// TIA Portal V19 export
DATA_BLOCK "RollformerLubr"   // DB140
// stored: InstanceOfName RollformerLubr_FB, InstanceOfType FB
"RollformerLubr_FB"
   // VAR_INPUT
   //    AreaInterface : "AreaInterface";
   // END_VAR
   // VAR_OUTPUT
   //    MachineInterface : "MachineInterface";
   // END_VAR
   // VAR
   //    Pump : "Lubr_Motor";
   //    Valves1 : "Lubr_Valve";
   //    Valves2 { S7_SetPoint := 'True'} : "Lubr_Valve";
   //    Valves3 { S7_SetPoint := 'True'} : "Lubr_Valve";
   // END_VAR
BEGIN
   AreaInterface.EStop := FALSE;
   AreaInterface.Man := TRUE;
   AreaInterface.Aut := FALSE;
   AreaInterface.Cycle := FALSE;
   AreaInterface.StopInPhase := FALSE;
   AreaInterface.StopProgrammed := FALSE;
   AreaInterface.RstAlarms := FALSE;
   AreaInterface.ManOneShot := FALSE;
   AreaInterface.AutOneShot := FALSE;
   AreaInterface.CycleOneShot := FALSE;
   AreaInterface.CheckAutReady := FALSE;
   MachineInterface.AutReady := FALSE;
   MachineInterface.Aborting := FALSE;
   MachineInterface.AckStopInPhase := FALSE;
   MachineInterface.AckStopProgrammed := FALSE;
   MachineInterface.MotionsStandStill := TRUE;
   MachineInterface.AlarmsPresence := FALSE;
   MachineInterface.WarningPresence := FALSE;
   Pump.DataIn.PbManualLubr := FALSE;
   Pump.DataIn.LubrRotationFbk := FALSE;
   Pump.DataIn.SensorLevel := TRUE;
   Pump.DataIn.MotorFdbkRunning := FALSE;
   Pump.DataIn.MotorThermalProtection := FALSE;
   Pump.ValveCycleTimeOut := T#5M;
   Pump.Simulation := FALSE;
   Pump.RunContactor := FALSE;
   Pump.Ctrl.RunReq := FALSE;
   Pump.Sts.OldValve := 1;
   Pump.Alarm.RotationFeedback := FALSE;
   Pump.Alarm.LowLevelLubrication := FALSE;
   Pump.Alarm.MotorAlr.ThermalProtection := FALSE;
   Pump.Alarm.MotorAlr.Feedback := FALSE;
   Pump.HMI.Alarm := FALSE;
   Pump.HMI.Running := FALSE;
   Pump.LubrInterface.Sts.PumpType := 0;
   Pump.LubrInterface.Sts.Running := FALSE;
   Pump.LubrInterface.Sts.Error := FALSE;
   Pump.LubrInterface.Ctrl.RstAlarms := FALSE;
   Pump.LubrInterface.Ctrl.WorkReq := FALSE;
   Pump.LubrInterface.ValveChain.ActualValve := 4;
   Pump.LubrInterface.ValveChain.MaxValve := 3;
   Pump.tonRotationON.PT := T#0MS;
   Pump.tonRotationON.IN := FALSE;
   Pump.tonRotationOFF.PT := T#0MS;
   Pump.tonRotationOFF.IN := FALSE;
   Pump.tonLowLevel.PT := T#0MS;
   Pump.tonLowLevel.IN := FALSE;
   Pump.ValveChianTimeOut.PT := T#5M;
   Pump.ValveChianTimeOut.IN := TRUE;
   Pump.LubrMotor.MotorCtrl.SafeStop := FALSE;
   Pump.LubrMotor.MotorCtrl.Rst := FALSE;
   Pump.LubrMotor.MotorCtrl.Run := FALSE;
   Pump.LubrMotor.ThermalProtection := FALSE;
   Pump.LubrMotor.FdbkRunning := FALSE;
   Pump.LubrMotor.FeedbackTimeout := T#500MS;
   Pump.LubrMotor.Simulation := FALSE;
   Pump.LubrMotor.MotorSts.AlarmPresence := FALSE;
   Pump.LubrMotor.MotorSts.RunPermitted := TRUE;
   Pump.LubrMotor.MotorSts.Running := FALSE;
   Pump.LubrMotor.Contactor := FALSE;
   Pump.LubrMotor.DelayContactorFeedbackON.PT := T#500MS;
   Pump.LubrMotor.DelayContactorFeedbackON.IN := FALSE;
   Pump.LubrMotor.Ctrl_RunContactor := FALSE;
   Valves1.AreaInterface.EStop := FALSE;
   Valves1.AreaInterface.Man := TRUE;
   Valves1.AreaInterface.Aut := FALSE;
   Valves1.AreaInterface.Cycle := FALSE;
   Valves1.AreaInterface.StopInPhase := FALSE;
   Valves1.AreaInterface.StopProgrammed := FALSE;
   Valves1.AreaInterface.RstAlarms := FALSE;
   Valves1.AreaInterface.ManOneShot := FALSE;
   Valves1.AreaInterface.AutOneShot := FALSE;
   Valves1.AreaInterface.CycleOneShot := FALSE;
   Valves1.AreaInterface.CheckAutReady := FALSE;
   Valves1.DataIn.PbStartLubr := FALSE;
   Valves1.DataIn.PbStopLubr := FALSE;
   Valves1.DataIn.CycleFbk := FALSE;
   Valves1.DataIn.ConnectorPlugged := TRUE;
   Valves1.CIn.LubrEnable := FALSE;
   Valves1.CIn.ActualPosition := 324862.052;
   Valves1.CIn.OperationDone := FALSE;
   Valves1.Config.WorkMode := 2;
   Valves1.Config.CounterMode := 0;
   Valves1.Config.ValveType := 1;
   Valves1.Config.ManualCmdTimeOut := T#5M;
   Valves1.Simulation := FALSE;
   Valves1.MachineInterface.AutReady := FALSE;
   Valves1.MachineInterface.Aborting := FALSE;
   Valves1.MachineInterface.AckStopInPhase := FALSE;
   Valves1.MachineInterface.AckStopProgrammed := FALSE;
   Valves1.MachineInterface.MotionsStandStill := TRUE;
   Valves1.MachineInterface.AlarmsPresence := FALSE;
   Valves1.MachineInterface.WarningPresence := FALSE;
   Valves1.COut.LubrReq := FALSE;
   Valves1.ValveCmd := FALSE;
   Valves1.Ctrl.ManualReq := FALSE;
   Valves1.Ctrl.AutomaticReq := FALSE;
   Valves1.Ctrl.LubrReq := FALSE;
   Valves1.Ctrl.ValveCmd := FALSE;
   Valves1.Sts.EstopDelayed := FALSE;
   Valves1.Sts.ValveEnabled := TRUE;
   Valves1.Sts.WorkEnable := TRUE;
   Valves1.Sts.CycleDone := FALSE;
   Valves1.Sts.LastFeed := 324862.052;
   Valves1.Sts.IsStandstill := TRUE;
   Valves1.Sts.AlarmsPresence := FALSE;
   Valves1.Sts.WarningsPresence := FALSE;
   Valves1.Alarm.CycleFeedback := FALSE;
   Valves1.Alarm.ConnectorNotPlugged := FALSE;
   Valves1.Alarm.ConfigError := FALSE;
   Valves1.Warning.SystemNotON := FALSE;
   Valves1.HMI.ManReq := FALSE;
   Valves1.HMI.AutoReq := FALSE;
   Valves1.HMI.Running := FALSE;
   Valves1.HMI.Alarm := FALSE;
   Valves1.HMI.ActualWorkTime := T#0MS;
   Valves1.tonEStopDelayed.PT := T#0MS;
   Valves1.tonEStopDelayed.IN := FALSE;
   Valves1.tonCycleDoneON.PT := T#0MS;
   Valves1.tonCycleDoneON.IN := FALSE;
   Valves1.tonCycleDoneOFF.PT := T#0MS;
   Valves1.tonCycleDoneOFF.IN := FALSE;
   Valves1.tonManualCycleReset.PT := T#5M;
   Valves1.tonManualCycleReset.IN := FALSE;
   Valves1.tonValveOn.PT := T#1S;
   Valves1.tonValveOn.IN := FALSE;
   Valves1.tonValveOff.PT := T#1S;
   Valves1.tonValveOff.IN := TRUE;
   Valves1.tonWorkTime.IN := FALSE;
   Valves1.tonWorkTime.ENA := FALSE;
   Valves1.tonWorkTime.PT := T#0MS;
   Valves1.tonWorkTime.Q := TRUE;
   Valves1.tonWorkTime.ET := T#0MS;
   Valves1.tonWorkTime.ton.PT := T#0MS;
   Valves1.tonWorkTime.ton.IN := FALSE;
   Valves1.tonWorkTime.LocalPT := T#0MS;
   Valves1.tonWorkTime.AuxSavePT := FALSE;
   Valves1.Aux_PbStartLubr := FALSE;
   Valves1.Pe_PbStartLubr := FALSE;
   Valves1.Aux_CyckeFkb := FALSE;
   Valves1.Pe_CycleFbk := FALSE;
   Valves1.Aux_OpDone := FALSE;
   Valves1.Pe_OpDone := FALSE;
   Valves1.Aux_ValveCount := TRUE;
   Valves1.Pe_ValveCount := FALSE;
   Valves2.AreaInterface.EStop := FALSE;
   Valves2.AreaInterface.Man := TRUE;
   Valves2.AreaInterface.Aut := FALSE;
   Valves2.AreaInterface.Cycle := FALSE;
   Valves2.AreaInterface.StopInPhase := FALSE;
   Valves2.AreaInterface.StopProgrammed := FALSE;
   Valves2.AreaInterface.RstAlarms := FALSE;
   Valves2.AreaInterface.ManOneShot := FALSE;
   Valves2.AreaInterface.AutOneShot := FALSE;
   Valves2.AreaInterface.CycleOneShot := FALSE;
   Valves2.AreaInterface.CheckAutReady := FALSE;
   Valves2.DataIn.PbStartLubr := FALSE;
   Valves2.DataIn.PbStopLubr := FALSE;
   Valves2.DataIn.CycleFbk := FALSE;
   Valves2.DataIn.ConnectorPlugged := TRUE;
   Valves2.CIn.LubrEnable := FALSE;
   Valves2.CIn.ActualPosition := 324862.052;
   Valves2.CIn.OperationDone := FALSE;
   Valves2.Config.WorkMode := 2;
   Valves2.Config.CounterMode := 0;
   Valves2.Config.ValveType := 1;
   Valves2.Config.ManualCmdTimeOut := T#5M;
   Valves2.Simulation := FALSE;
   Valves2.MachineInterface.AutReady := FALSE;
   Valves2.MachineInterface.Aborting := FALSE;
   Valves2.MachineInterface.AckStopInPhase := FALSE;
   Valves2.MachineInterface.AckStopProgrammed := FALSE;
   Valves2.MachineInterface.MotionsStandStill := TRUE;
   Valves2.MachineInterface.AlarmsPresence := FALSE;
   Valves2.MachineInterface.WarningPresence := FALSE;
   Valves2.COut.LubrReq := FALSE;
   Valves2.ValveCmd := FALSE;
   Valves2.Ctrl.ManualReq := FALSE;
   Valves2.Ctrl.AutomaticReq := FALSE;
   Valves2.Ctrl.LubrReq := FALSE;
   Valves2.Ctrl.ValveCmd := FALSE;
   Valves2.Sts.EstopDelayed := FALSE;
   Valves2.Sts.ValveEnabled := TRUE;
   Valves2.Sts.WorkEnable := TRUE;
   Valves2.Sts.CycleDone := FALSE;
   Valves2.Sts.LastFeed := 324862.052;
   Valves2.Sts.IsStandstill := TRUE;
   Valves2.Sts.AlarmsPresence := FALSE;
   Valves2.Sts.WarningsPresence := FALSE;
   Valves2.Alarm.CycleFeedback := FALSE;
   Valves2.Alarm.ConnectorNotPlugged := FALSE;
   Valves2.Alarm.ConfigError := FALSE;
   Valves2.Warning.SystemNotON := FALSE;
   Valves2.HMI.ManReq := FALSE;
   Valves2.HMI.AutoReq := FALSE;
   Valves2.HMI.Running := FALSE;
   Valves2.HMI.Alarm := FALSE;
   Valves2.HMI.ActualWorkTime := T#0MS;
   Valves2.tonEStopDelayed.PT := T#0MS;
   Valves2.tonEStopDelayed.IN := FALSE;
   Valves2.tonCycleDoneON.PT := T#0MS;
   Valves2.tonCycleDoneON.IN := FALSE;
   Valves2.tonCycleDoneOFF.PT := T#0MS;
   Valves2.tonCycleDoneOFF.IN := FALSE;
   Valves2.tonManualCycleReset.PT := T#0MS;
   Valves2.tonManualCycleReset.IN := FALSE;
   Valves2.tonValveOn.PT := T#1S;
   Valves2.tonValveOn.IN := FALSE;
   Valves2.tonValveOff.PT := T#1S;
   Valves2.tonValveOff.IN := TRUE;
   Valves2.tonWorkTime.IN := FALSE;
   Valves2.tonWorkTime.ENA := FALSE;
   Valves2.tonWorkTime.PT := T#0MS;
   Valves2.tonWorkTime.Q := TRUE;
   Valves2.tonWorkTime.ET := T#0MS;
   Valves2.tonWorkTime.ton.PT := T#0MS;
   Valves2.tonWorkTime.ton.IN := FALSE;
   Valves2.tonWorkTime.LocalPT := T#0MS;
   Valves2.tonWorkTime.AuxSavePT := FALSE;
   Valves2.Aux_PbStartLubr := FALSE;
   Valves2.Pe_PbStartLubr := FALSE;
   Valves2.Aux_CyckeFkb := FALSE;
   Valves2.Pe_CycleFbk := FALSE;
   Valves2.Aux_OpDone := FALSE;
   Valves2.Pe_OpDone := FALSE;
   Valves2.Aux_ValveCount := TRUE;
   Valves2.Pe_ValveCount := FALSE;
   Valves3.AreaInterface.EStop := FALSE;
   Valves3.AreaInterface.Man := TRUE;
   Valves3.AreaInterface.Aut := FALSE;
   Valves3.AreaInterface.Cycle := FALSE;
   Valves3.AreaInterface.StopInPhase := FALSE;
   Valves3.AreaInterface.StopProgrammed := FALSE;
   Valves3.AreaInterface.RstAlarms := FALSE;
   Valves3.AreaInterface.ManOneShot := FALSE;
   Valves3.AreaInterface.AutOneShot := FALSE;
   Valves3.AreaInterface.CycleOneShot := FALSE;
   Valves3.AreaInterface.CheckAutReady := FALSE;
   Valves3.DataIn.PbStartLubr := FALSE;
   Valves3.DataIn.PbStopLubr := FALSE;
   Valves3.DataIn.CycleFbk := FALSE;
   Valves3.DataIn.ConnectorPlugged := TRUE;
   Valves3.CIn.LubrEnable := FALSE;
   Valves3.CIn.ActualPosition := 324862.052;
   Valves3.CIn.OperationDone := FALSE;
   Valves3.Config.WorkMode := 2;
   Valves3.Config.CounterMode := 0;
   Valves3.Config.ValveType := 1;
   Valves3.Config.ManualCmdTimeOut := T#5M;
   Valves3.Simulation := FALSE;
   Valves3.MachineInterface.AutReady := FALSE;
   Valves3.MachineInterface.Aborting := FALSE;
   Valves3.MachineInterface.AckStopInPhase := FALSE;
   Valves3.MachineInterface.AckStopProgrammed := FALSE;
   Valves3.MachineInterface.MotionsStandStill := TRUE;
   Valves3.MachineInterface.AlarmsPresence := FALSE;
   Valves3.MachineInterface.WarningPresence := FALSE;
   Valves3.COut.LubrReq := FALSE;
   Valves3.ValveCmd := FALSE;
   Valves3.Ctrl.ManualReq := FALSE;
   Valves3.Ctrl.AutomaticReq := FALSE;
   Valves3.Ctrl.LubrReq := FALSE;
   Valves3.Ctrl.ValveCmd := FALSE;
   Valves3.Sts.EstopDelayed := FALSE;
   Valves3.Sts.ValveEnabled := TRUE;
   Valves3.Sts.WorkEnable := TRUE;
   Valves3.Sts.CycleDone := FALSE;
   Valves3.Sts.LastFeed := 324862.052;
   Valves3.Sts.IsStandstill := TRUE;
   Valves3.Sts.AlarmsPresence := FALSE;
   Valves3.Sts.WarningsPresence := FALSE;
   Valves3.Alarm.CycleFeedback := FALSE;
   Valves3.Alarm.ConnectorNotPlugged := FALSE;
   Valves3.Alarm.ConfigError := FALSE;
   Valves3.Warning.SystemNotON := FALSE;
   Valves3.HMI.ManReq := FALSE;
   Valves3.HMI.AutoReq := FALSE;
   Valves3.HMI.Running := FALSE;
   Valves3.HMI.Alarm := FALSE;
   Valves3.HMI.ActualWorkTime := T#0MS;
   Valves3.tonEStopDelayed.PT := T#0MS;
   Valves3.tonEStopDelayed.IN := FALSE;
   Valves3.tonCycleDoneON.PT := T#0MS;
   Valves3.tonCycleDoneON.IN := FALSE;
   Valves3.tonCycleDoneOFF.PT := T#0MS;
   Valves3.tonCycleDoneOFF.IN := FALSE;
   Valves3.tonManualCycleReset.PT := T#0MS;
   Valves3.tonManualCycleReset.IN := FALSE;
   Valves3.tonValveOn.PT := T#1S;
   Valves3.tonValveOn.IN := FALSE;
   Valves3.tonValveOff.PT := T#1S;
   Valves3.tonValveOff.IN := TRUE;
   Valves3.tonWorkTime.IN := FALSE;
   Valves3.tonWorkTime.ENA := FALSE;
   Valves3.tonWorkTime.PT := T#0MS;
   Valves3.tonWorkTime.Q := TRUE;
   Valves3.tonWorkTime.ET := T#0MS;
   Valves3.tonWorkTime.ton.PT := T#0MS;
   Valves3.tonWorkTime.ton.IN := FALSE;
   Valves3.tonWorkTime.LocalPT := T#0MS;
   Valves3.tonWorkTime.AuxSavePT := FALSE;
   Valves3.Aux_PbStartLubr := FALSE;
   Valves3.Pe_PbStartLubr := FALSE;
   Valves3.Aux_CyckeFkb := FALSE;
   Valves3.Pe_CycleFbk := FALSE;
   Valves3.Aux_OpDone := FALSE;
   Valves3.Pe_OpDone := FALSE;
   Valves3.Aux_ValveCount := TRUE;
   Valves3.Pe_ValveCount := FALSE;
END_DATA_BLOCK
